FUNCTION_BLOCK fb_IO_Basic
VAR_INPUT
END_VAR
VAR_OUTPUT
END_VAR
VAR
END_VAR

END_FUNCTION_BLOCK

(* stored: Version 1.1.0.1, ProductVersion 3.1.4024.3
   POU fb_IO_Basic: Id {b9dc89ab-8c33-4bb3-8945-785bc1d3fd3f}, SpecialFunc None *)
